(* Logix 5000 project; controller cal1615 1756-L62 rev 20.19; software revision 20.05; part 31 of 82 *)
(* tags used below, declared in another part *)
   FAULT : BOOL;   // Fault AFI
   p01_param_oven_timer_presets : DINT[32];   // System Parameter Oven Timer Presets
   p01_param_process_air_hl : REAL;   // Machine Parameter Process Air High Limit
   p01_sys_enc : SYS_ENC;   // System Encoder
   p01_sys_lc : Limit_Clamp;   // Zone 1 Misc Control Limit Clamp
   p01r09_pb_global_reset : BOOL;   // System Modes PB: Global Fault Reset
   p01r11 : routine;   // System Timer Presets
   p02_real_from_hmi : hmi_real;   // MOP HMI Iface Real from HMI
   p12r31_timer_warning : TIMER[5];   // Zone 2 Exhaust VFD Waringing Timer
   p12r32_timer_warning : TIMER[5];   // Zone 2 Supply VFD Warning Timer
   p13_di_exh_flow_ok : BOOL;   // Zone 3 Digital Input Exhaust Flow OK
   p13_di_recirc_flow_ok : BOOL;   // Zone 3 Digital Input Recirc Flow OK
   p13_param_fast_to_soak : REAL;   // Zone 3 Parameter Fast to Soak Control
   p13_param_lfl_hhl : REAL;   // Zone 3 Parameter High High Lower Flash Limit
   p13_param_lfl_hl : REAL;   // Zone 3 Parameter High LFL Limit
   p13_param_pid1_ff : REAL;   // Zone 3 Parameter Fast PID Bias
   p13_param_pid1_kd : REAL;   // Zone 3 Parameter Fast PID Derivative Gain
   p13_param_pid1_ki : REAL;   // Zone 3 Parameter Fast PID Integral Gain
   p13_param_pid1_kp : REAL;   // Zone 3 Parameter Fast PID Proportional Gain
   p13_param_pid2_ff : REAL;   // Zone 3 Parameter Auto PID Bias
   p13_param_pid2_kd : REAL;   // Zone 3 Parameter Auto PID Derivative Gain
   p13_param_pid2_ki : REAL;   // Zone 3 Parameter Auto PID Integral Gain
   p13_param_pid2_kp : REAL;   // Zone 3 Parameter Auto PID Proportional Gain
   p13_param_shutdown_temp : REAL;   // Zone 3 Parameter Zone Shutdown Temperature
   p13_param_soak_to_fast : REAL;   // Zone 3 Parameter Soak to Fast Control
   p13_param_tc01_dev : REAL;   // Zone 3 Parameter Oven Temperature Deviation from Setpoint
   p13_param_tc01_hl : REAL;   // Zone 3 Parameter Process Air High Limit
   p13_param_tc01z : REAL;   // Zone 3 Parameter Process Temperature Zero Offset
   p13_param_tc02z : REAL;   // Zone 3 Parameter SupplyTemperature Zero Offset
   p13_param_zone_pressure : REAL;   // Zone 3 Parameter High Pressure LImit
   p13r01 : routine;   // Zone 3 Main
   p13r02_timer_safe_temp : TIMER[2];   // Zone 3 Misc Control Chamber SafeTemperature Dwell
   p13r02_timer_warning : TIMER[4];   // Zone 3 Misc Control Warning Delay
   p13r09 : routine;   // Zone 3 Modes
   p13r09_timer_fault : TIMER[4];   // Zone 3 Modes Fault Delay
   p13r09_timer_warning : TIMER[8];   // Zone 3 Modes Warning Delay
   p13r10 : routine;   // Zone 3
   p13r10_timer_fault : TIMER[4];   // Zone 3 Fault Delay
   p13r10_timer_warning : TIMER[4];   // Zone 3 Warning Delay
   p13r20 : routine;   // Zone 3 Temp Sequence
   p13r20_state : DINT;   // Zone 3 Temperature Control State
   p13r20_status : DINT;   // Zone 3 Temperature Control Sequence Status
   p13r20_timer_fault : TIMER[4];   // Zone 3 Temp Sequence Fault Delay
   p13r20_timer_state_11 : TIMER;   // Zone 3 Temp Sequence State 11 Dwell
   p13r20_timer_state_3 : TIMER;   // Zone 3 Temperature Control State 3 Dwell
   p13r20_timer_state_4 : TIMER;   // Zone 3 Temp Sequence State 4 Dwell
   p13r20_timer_state_7 : TIMER;   // Zone 3 Temp Sequence State 7 Dwell
   p13r20_timer_warning : TIMER[4];   // Zone 3 Temp Sequence Warning Delay
   p13r30_cv_man_sp : REAL;   // Zone 3 Temperature Control Manual Heat Control Valve Setpoint
   p13r30_request_cool : BOOL;   // Zone 3 Temperature Control Request Cooling
   p13r30_request_manual : BOOL;   // Zone 3 Temperature Control Request Manual Control
   p13r30_temp_deviation_setpoint : DINT;
   p13r30_timer_fault : TIMER[16];   // Zone 3 Temperature Control Fault Delay
   p13r30_timer_warning : TIMER[12];   // Zone 3 Temperature Control Warning Delay
   p13r31_timer_fault : TIMER[5];   // Zone 3 Exhaust VFD Fault Timer
   p13r31_timer_warning : TIMER[5];   // Zone 3 Exhaust VFD Waringing Timer
   p13r32_timer_fault : TIMER[5];   // Zone 3 Recirc VFD Fault Timer
   p13r32_timer_warning : TIMER[5];   // Zone 3 Supply VFD Warning Timer
(* P13_Zone_3, continued *)

ROUTINE R09_Modes   (* ladder *)
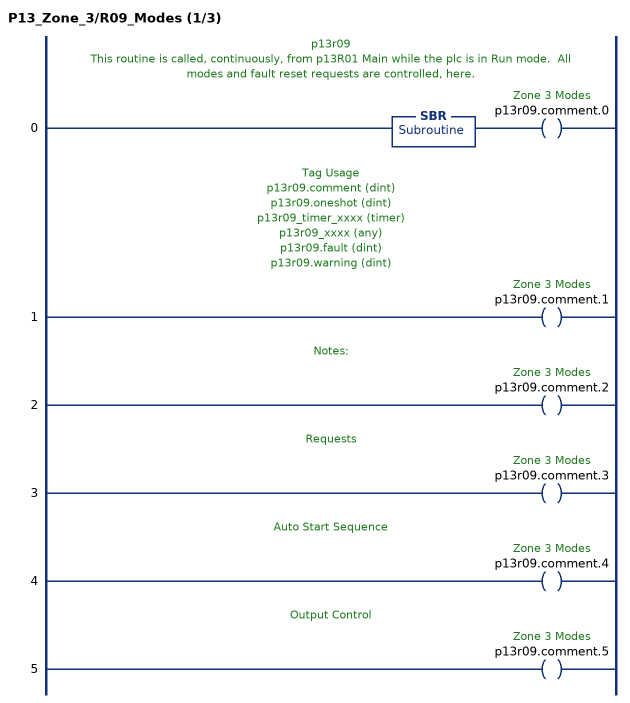
   // p13r09
   // This routine is called, continuously, from p13R01 Main while the plc is in Run mode.  All modes and fault reset requests are controlled, here.
   0: SBR()OTE(p13r09.comment.0);
   // Tag Usage
   // p13r09.comment (dint)
   // p13r09.oneshot (dint)
   // p13r09_timer_xxxx (timer)
   // p13r09_xxxx (any)
   // p13r09.fault (dint)
   // p13r09.warning (dint)
   1: OTE(p13r09.comment.1);
   // Notes:
   2: OTE(p13r09.comment.2);
   // Requests
   3: OTE(p13r09.comment.3);
   // Auto Start Sequence
   4: OTE(p13r09.comment.4);
   // Output Control
   5: OTE(p13r09.comment.5);
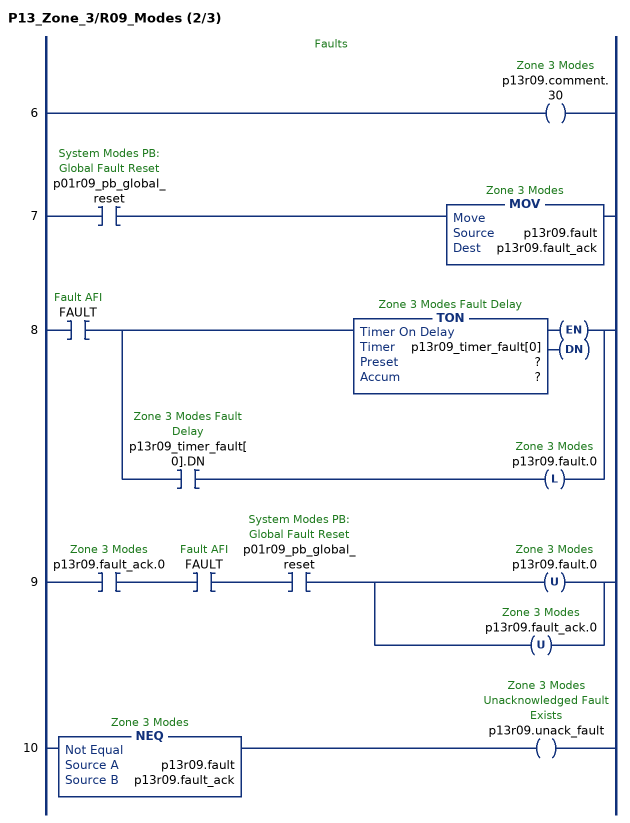
   // Faults
   6: OTE(p13r09.comment.30);
   7: XIC(p01r09_pb_global_reset)MOV(p13r09.fault,p13r09.fault_ack);
   8: XIC(FAULT)[TON(p13r09_timer_fault[0],?,?) ,XIC(p13r09_timer_fault[0].DN) OTL(p13r09.fault.0) ];
   9: XIC(p13r09.fault_ack.0)XIC(FAULT)XIC(p01r09_pb_global_reset)[OTU(p13r09.fault.0) ,OTU(p13r09.fault_ack.0) ];
   10: NEQ(p13r09.fault,p13r09.fault_ack)OTE(p13r09.unack_fault);
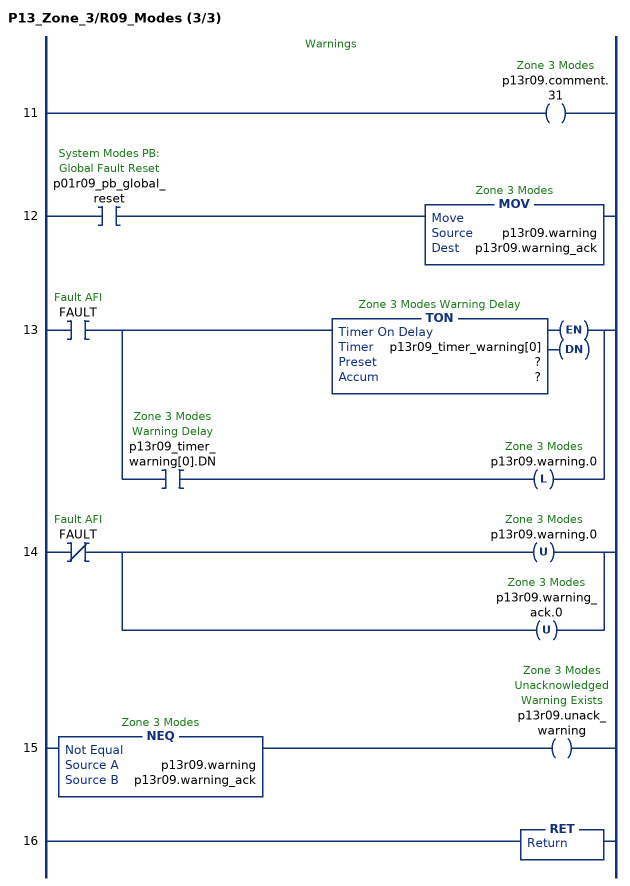
   // Warnings
   11: OTE(p13r09.comment.31);
   12: XIC(p01r09_pb_global_reset)MOV(p13r09.warning,p13r09.warning_ack);
   13: XIC(FAULT)[TON(p13r09_timer_warning[0],?,?) ,XIC(p13r09_timer_warning[0].DN) OTL(p13r09.warning.0) ];
   14: XIO(FAULT)[OTU(p13r09.warning.0) ,OTU(p13r09.warning_ack.0) ];
   15: NEQ(p13r09.warning,p13r09.warning_ack)OTE(p13r09.unack_warning);
   16: RET();
END_ROUTINE

ROUTINE R10_Parameters   (* ladder *)
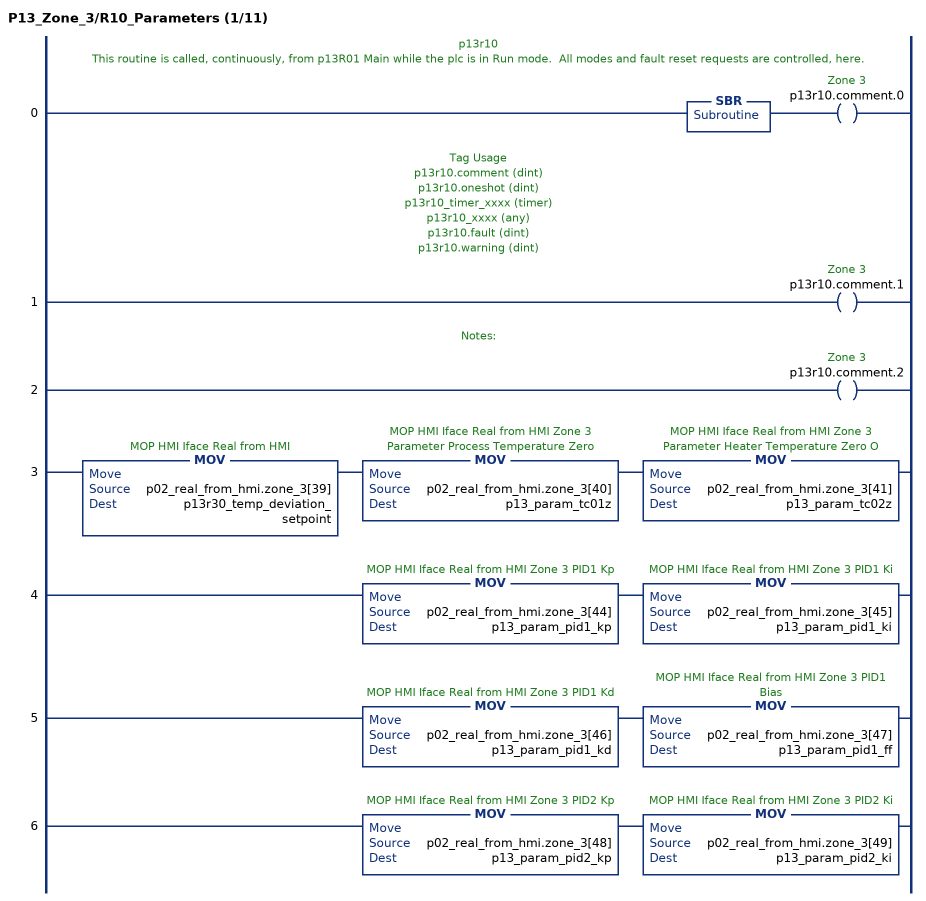
   // p13r10
   // This routine is called, continuously, from p13R01 Main while the plc is in Run mode.  All modes and fault reset requests are controlled, here.
   0: SBR()OTE(p13r10.comment.0);
   // Tag Usage
   // p13r10.comment (dint)
   // p13r10.oneshot (dint)
   // p13r10_timer_xxxx (timer)
   // p13r10_xxxx (any)
   // p13r10.fault (dint)
   // p13r10.warning (dint)
   1: OTE(p13r10.comment.1);
   // Notes:
   2: OTE(p13r10.comment.2);
   3: MOV(p02_real_from_hmi.zone_3[39],p13r30_temp_deviation_setpoint)MOV(p02_real_from_hmi.zone_3[40],p13_param_tc01z)MOV(p02_real_from_hmi.zone_3[41],p13_param_tc02z);
   4: MOV(p02_real_from_hmi.zone_3[44],p13_param_pid1_kp)MOV(p02_real_from_hmi.zone_3[45],p13_param_pid1_ki);
   5: MOV(p02_real_from_hmi.zone_3[46],p13_param_pid1_kd)MOV(p02_real_from_hmi.zone_3[47],p13_param_pid1_ff);
   6: MOV(p02_real_from_hmi.zone_3[48],p13_param_pid2_kp)MOV(p02_real_from_hmi.zone_3[49],p13_param_pid2_ki);
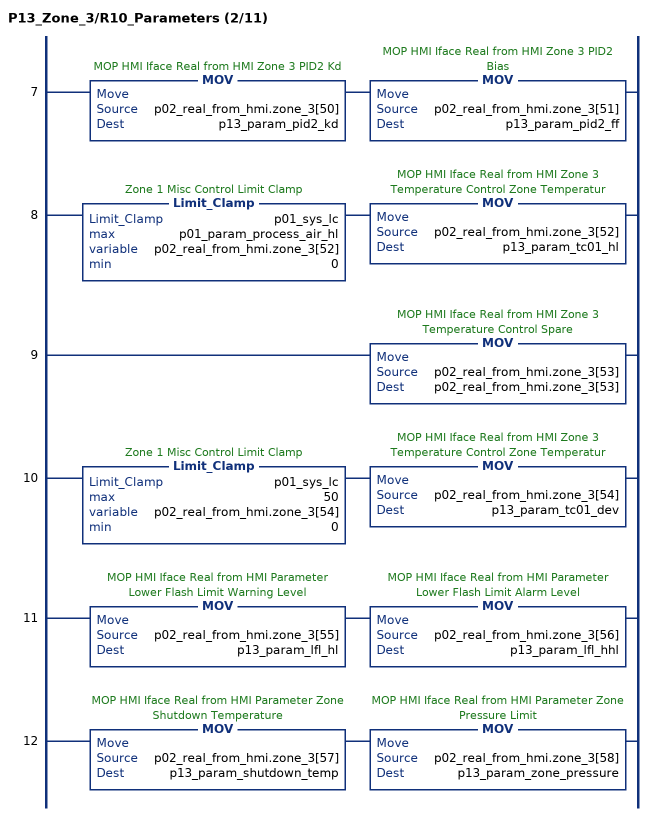
   7: MOV(p02_real_from_hmi.zone_3[50],p13_param_pid2_kd)MOV(p02_real_from_hmi.zone_3[51],p13_param_pid2_ff);
   8: Limit_Clamp(p01_sys_lc,p01_param_process_air_hl,p02_real_from_hmi.zone_3[52],0)MOV(p02_real_from_hmi.zone_3[52],p13_param_tc01_hl);
   9: MOV(p02_real_from_hmi.zone_3[53],p02_real_from_hmi.zone_3[53]);
   10: Limit_Clamp(p01_sys_lc,50,p02_real_from_hmi.zone_3[54],0)MOV(p02_real_from_hmi.zone_3[54],p13_param_tc01_dev);
   11: MOV(p02_real_from_hmi.zone_3[55],p13_param_lfl_hl)MOV(p02_real_from_hmi.zone_3[56],p13_param_lfl_hhl);
   12: MOV(p02_real_from_hmi.zone_3[57],p13_param_shutdown_temp)MOV(p02_real_from_hmi.zone_3[58],p13_param_zone_pressure);
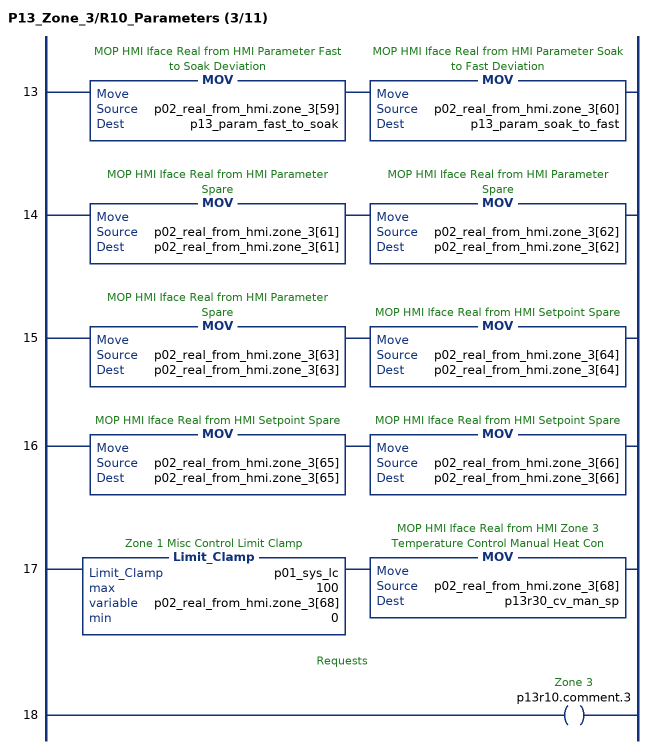
   13: MOV(p02_real_from_hmi.zone_3[59],p13_param_fast_to_soak)MOV(p02_real_from_hmi.zone_3[60],p13_param_soak_to_fast);
   14: MOV(p02_real_from_hmi.zone_3[61],p02_real_from_hmi.zone_3[61])MOV(p02_real_from_hmi.zone_3[62],p02_real_from_hmi.zone_3[62]);
   15: MOV(p02_real_from_hmi.zone_3[63],p02_real_from_hmi.zone_3[63])MOV(p02_real_from_hmi.zone_3[64],p02_real_from_hmi.zone_3[64]);
   16: MOV(p02_real_from_hmi.zone_3[65],p02_real_from_hmi.zone_3[65])MOV(p02_real_from_hmi.zone_3[66],p02_real_from_hmi.zone_3[66]);
   17: Limit_Clamp(p01_sys_lc,100,p02_real_from_hmi.zone_3[68],0)MOV(p02_real_from_hmi.zone_3[68],p13r30_cv_man_sp);
   // Requests
   18: OTE(p13r10.comment.3);
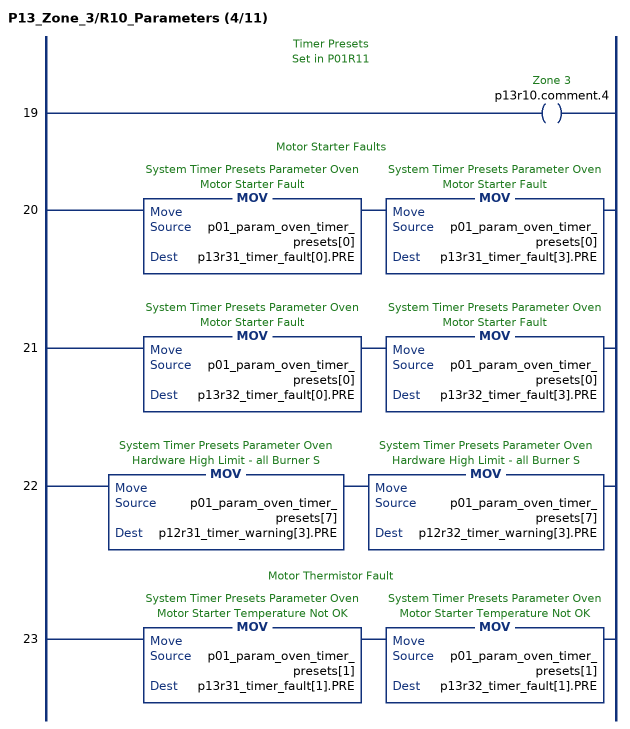
   // Timer Presets
   // Set in P01R11
   19: OTE(p13r10.comment.4);
   // Motor Starter Faults
   20: MOV(p01_param_oven_timer_presets[0],p13r31_timer_fault[0].PRE)MOV(p01_param_oven_timer_presets[0],p13r31_timer_fault[3].PRE);
   21: MOV(p01_param_oven_timer_presets[0],p13r32_timer_fault[0].PRE)MOV(p01_param_oven_timer_presets[0],p13r32_timer_fault[3].PRE);
   22: MOV(p01_param_oven_timer_presets[7],p12r31_timer_warning[3].PRE)MOV(p01_param_oven_timer_presets[7],p12r32_timer_warning[3].PRE);
   // Motor Thermistor Fault
   23: MOV(p01_param_oven_timer_presets[1],p13r31_timer_fault[1].PRE)MOV(p01_param_oven_timer_presets[1],p13r32_timer_fault[1].PRE);
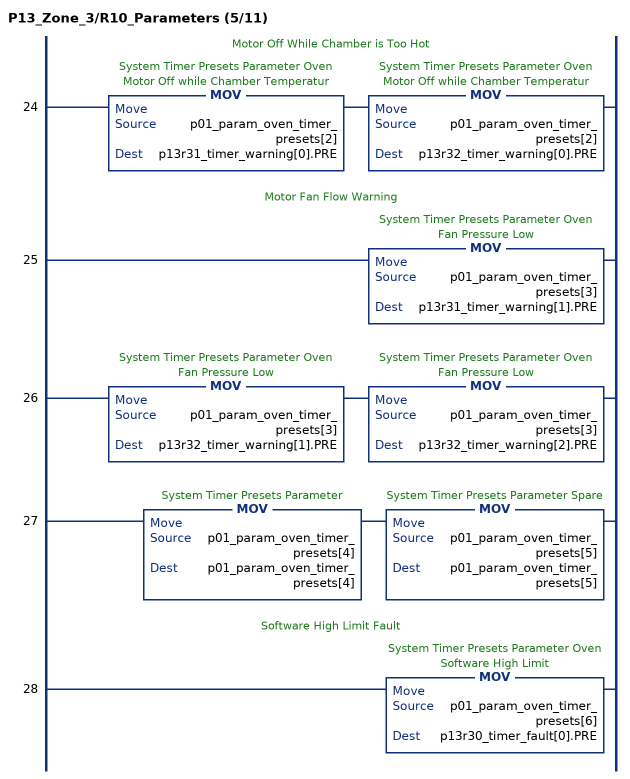
   // Motor Off While Chamber is Too Hot
   24: MOV(p01_param_oven_timer_presets[2],p13r31_timer_warning[0].PRE)MOV(p01_param_oven_timer_presets[2],p13r32_timer_warning[0].PRE);
   // Motor Fan Flow Warning
   25: MOV(p01_param_oven_timer_presets[3],p13r31_timer_warning[1].PRE);
   26: MOV(p01_param_oven_timer_presets[3],p13r32_timer_warning[1].PRE)MOV(p01_param_oven_timer_presets[3],p13r32_timer_warning[2].PRE);
   27: MOV(p01_param_oven_timer_presets[4],p01_param_oven_timer_presets[4])MOV(p01_param_oven_timer_presets[5],p01_param_oven_timer_presets[5]);
   // Software High Limit Fault
   28: MOV(p01_param_oven_timer_presets[6],p13r30_timer_fault[0].PRE);
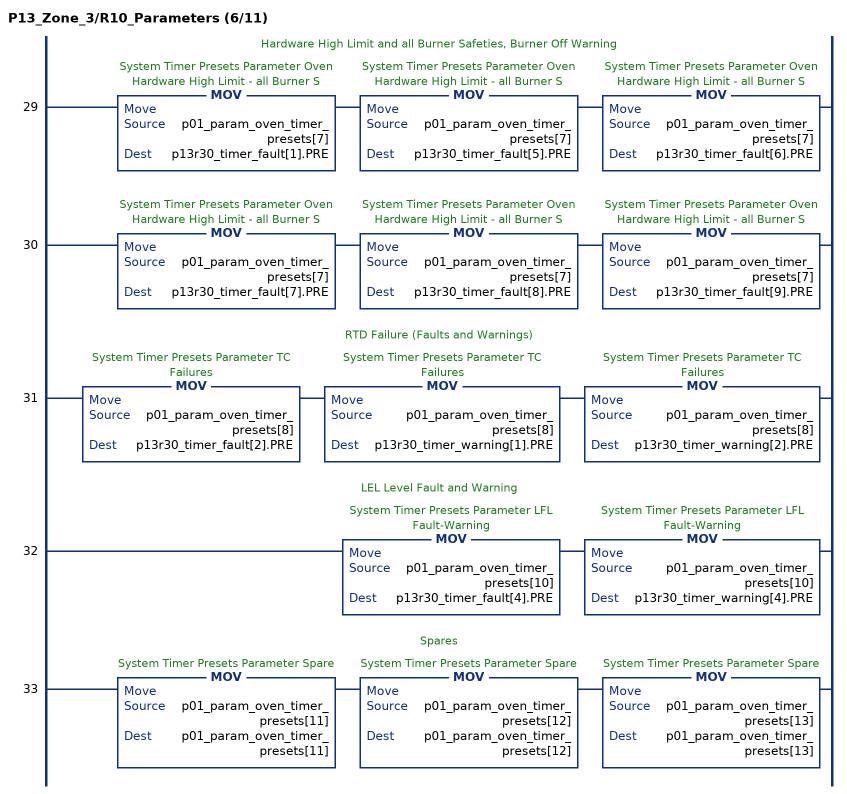
   // Hardware High Limit and all Burner Safeties, Burner Off Warning
   29: MOV(p01_param_oven_timer_presets[7],p13r30_timer_fault[1].PRE)MOV(p01_param_oven_timer_presets[7],p13r30_timer_fault[5].PRE)MOV(p01_param_oven_timer_presets[7],p13r30_timer_fault[6].PRE);
   30: MOV(p01_param_oven_timer_presets[7],p13r30_timer_fault[7].PRE)MOV(p01_param_oven_timer_presets[7],p13r30_timer_fault[8].PRE)MOV(p01_param_oven_timer_presets[7],p13r30_timer_fault[9].PRE);
   // RTD Failure (Faults and Warnings)
   31: MOV(p01_param_oven_timer_presets[8],p13r30_timer_fault[2].PRE)MOV(p01_param_oven_timer_presets[8],p13r30_timer_warning[1].PRE)MOV(p01_param_oven_timer_presets[8],p13r30_timer_warning[2].PRE);
   // LEL Level Fault and Warning
   32: MOV(p01_param_oven_timer_presets[10],p13r30_timer_fault[4].PRE)MOV(p01_param_oven_timer_presets[10],p13r30_timer_warning[4].PRE);
   // Spares
   33: MOV(p01_param_oven_timer_presets[11],p01_param_oven_timer_presets[11])MOV(p01_param_oven_timer_presets[12],p01_param_oven_timer_presets[12])MOV(p01_param_oven_timer_presets[13],p01_param_oven_timer_presets[13]);
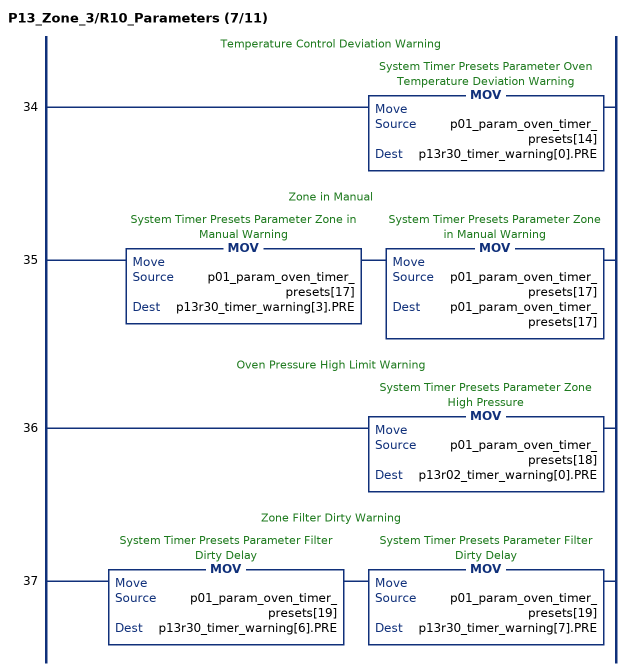
   // Temperature Control Deviation Warning
   34: MOV(p01_param_oven_timer_presets[14],p13r30_timer_warning[0].PRE);
   // Zone in Manual
   35: MOV(p01_param_oven_timer_presets[17],p13r30_timer_warning[3].PRE)MOV(p01_param_oven_timer_presets[17],p01_param_oven_timer_presets[17]);
   // Oven Pressure High Limit Warning
   36: MOV(p01_param_oven_timer_presets[18],p13r02_timer_warning[0].PRE);
   // Zone Filter Dirty Warning
   37: MOV(p01_param_oven_timer_presets[19],p13r30_timer_warning[6].PRE)MOV(p01_param_oven_timer_presets[19],p13r30_timer_warning[7].PRE);
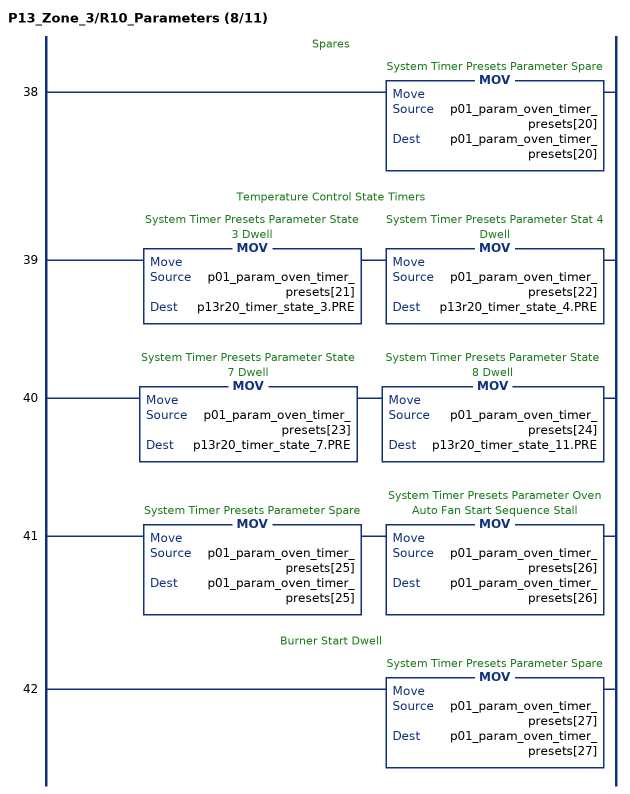
   // Spares
   38: MOV(p01_param_oven_timer_presets[20],p01_param_oven_timer_presets[20]);
   // Temperature Control State Timers
   39: MOV(p01_param_oven_timer_presets[21],p13r20_timer_state_3.PRE)MOV(p01_param_oven_timer_presets[22],p13r20_timer_state_4.PRE);
   40: MOV(p01_param_oven_timer_presets[23],p13r20_timer_state_7.PRE)MOV(p01_param_oven_timer_presets[24],p13r20_timer_state_11.PRE);
   41: MOV(p01_param_oven_timer_presets[25],p01_param_oven_timer_presets[25])MOV(p01_param_oven_timer_presets[26],p01_param_oven_timer_presets[26]);
   // Burner Start Dwell
   42: MOV(p01_param_oven_timer_presets[27],p01_param_oven_timer_presets[27]);
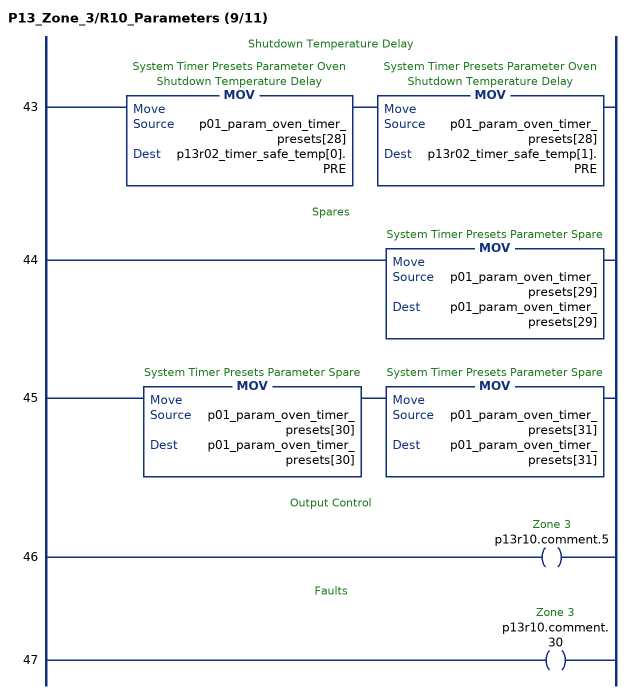
   // Shutdown Temperature Delay
   43: MOV(p01_param_oven_timer_presets[28],p13r02_timer_safe_temp[0].PRE)MOV(p01_param_oven_timer_presets[28],p13r02_timer_safe_temp[1].PRE);
   // Spares
   44: MOV(p01_param_oven_timer_presets[29],p01_param_oven_timer_presets[29]);
   45: MOV(p01_param_oven_timer_presets[30],p01_param_oven_timer_presets[30])MOV(p01_param_oven_timer_presets[31],p01_param_oven_timer_presets[31]);
   // Output Control
   46: OTE(p13r10.comment.5);
   // Faults
   47: OTE(p13r10.comment.30);
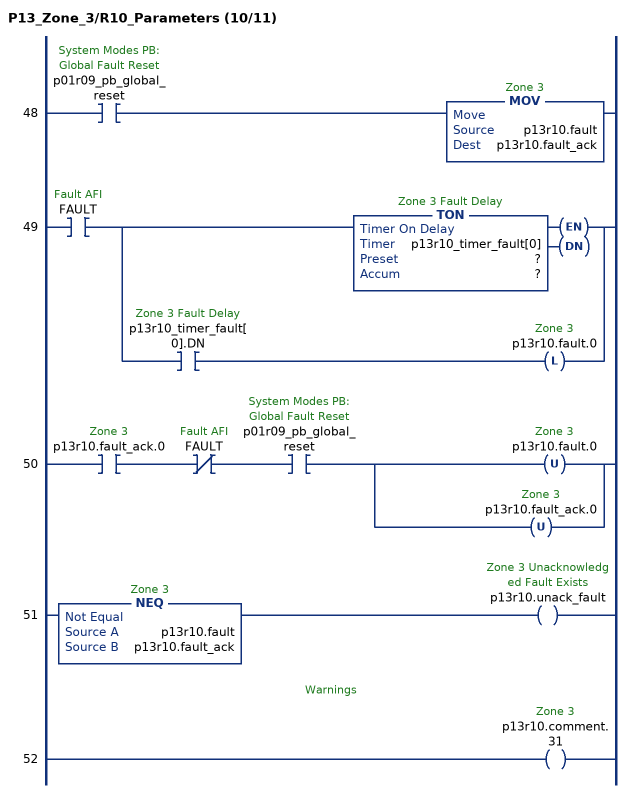
   48: XIC(p01r09_pb_global_reset)MOV(p13r10.fault,p13r10.fault_ack);
   49: XIC(FAULT)[TON(p13r10_timer_fault[0],?,?) ,XIC(p13r10_timer_fault[0].DN) OTL(p13r10.fault.0) ];
   50: XIC(p13r10.fault_ack.0)XIO(FAULT)XIC(p01r09_pb_global_reset)[OTU(p13r10.fault.0) ,OTU(p13r10.fault_ack.0) ];
   51: NEQ(p13r10.fault,p13r10.fault_ack)OTE(p13r10.unack_fault);
   // Warnings
   52: OTE(p13r10.comment.31);
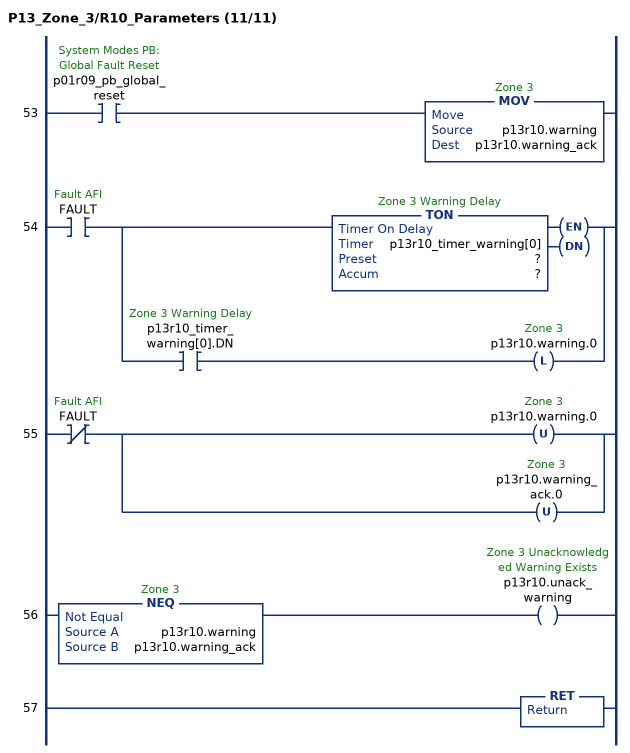
   53: XIC(p01r09_pb_global_reset)MOV(p13r10.warning,p13r10.warning_ack);
   54: XIC(FAULT)[TON(p13r10_timer_warning[0],?,?) ,XIC(p13r10_timer_warning[0].DN) OTL(p13r10.warning.0) ];
   55: XIO(FAULT)[OTU(p13r10.warning.0) ,OTU(p13r10.warning_ack.0) ];
   56: NEQ(p13r10.warning,p13r10.warning_ack)OTE(p13r10.unack_warning);
   57: RET();
END_ROUTINE

ROUTINE R20_Temp_Sequence   (* ladder *)
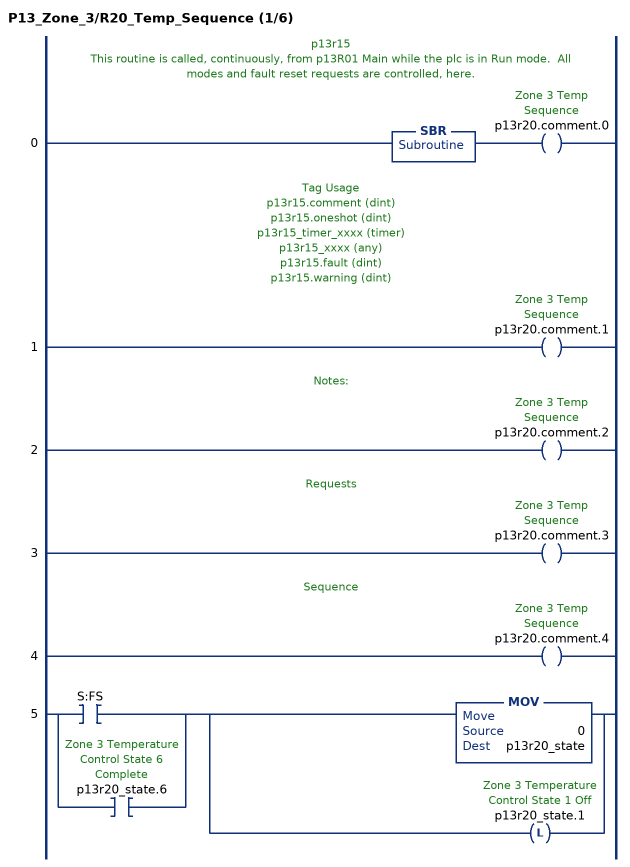
   // p13r15
   // This routine is called, continuously, from p13R01 Main while the plc is in Run mode.  All modes and fault reset requests are controlled, here.
   0: SBR()OTE(p13r20.comment.0);
   // Tag Usage
   // p13r15.comment (dint)
   // p13r15.oneshot (dint)
   // p13r15_timer_xxxx (timer)
   // p13r15_xxxx (any)
   // p13r15.fault (dint)
   // p13r15.warning (dint)
   1: OTE(p13r20.comment.1);
   // Notes:
   2: OTE(p13r20.comment.2);
   // Requests
   3: OTE(p13r20.comment.3);
   // Sequence
   4: OTE(p13r20.comment.4);
   5: [XIC(S:FS) ,XIC(p13r20_state.6) ][MOV(0,p13r20_state) ,OTL(p13r20_state.1) ];
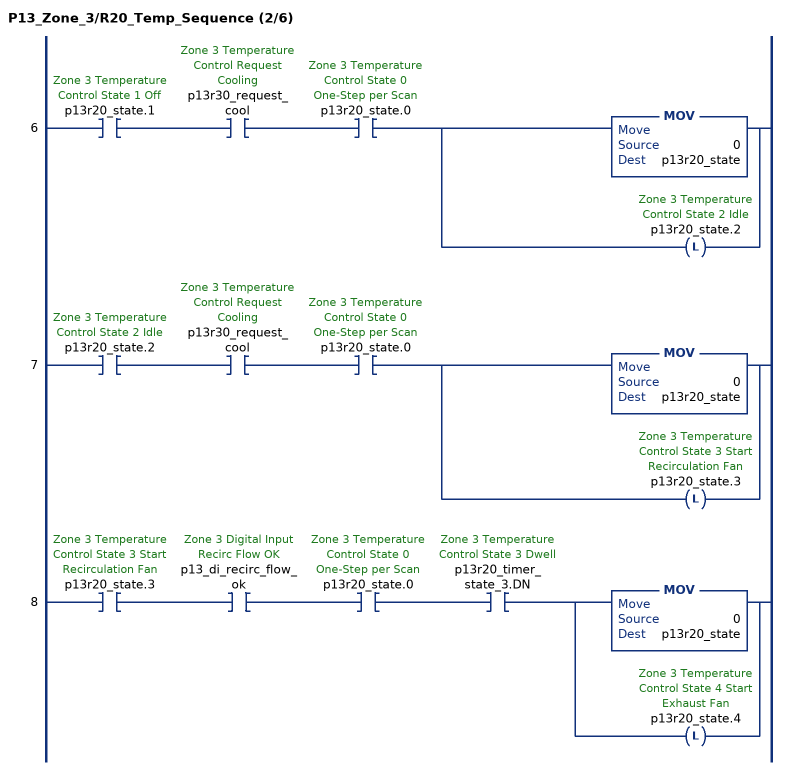
   6: XIC(p13r20_state.1)XIC(p13r30_request_cool)XIC(p13r20_state.0)[MOV(0,p13r20_state) ,OTL(p13r20_state.2) ];
   7: XIC(p13r20_state.2)XIC(p13r30_request_cool)XIC(p13r20_state.0)[MOV(0,p13r20_state) ,OTL(p13r20_state.3) ];
   8: XIC(p13r20_state.3)XIC(p13_di_recirc_flow_ok)XIC(p13r20_state.0)XIC(p13r20_timer_state_3.DN)[MOV(0,p13r20_state) ,OTL(p13r20_state.4) ];
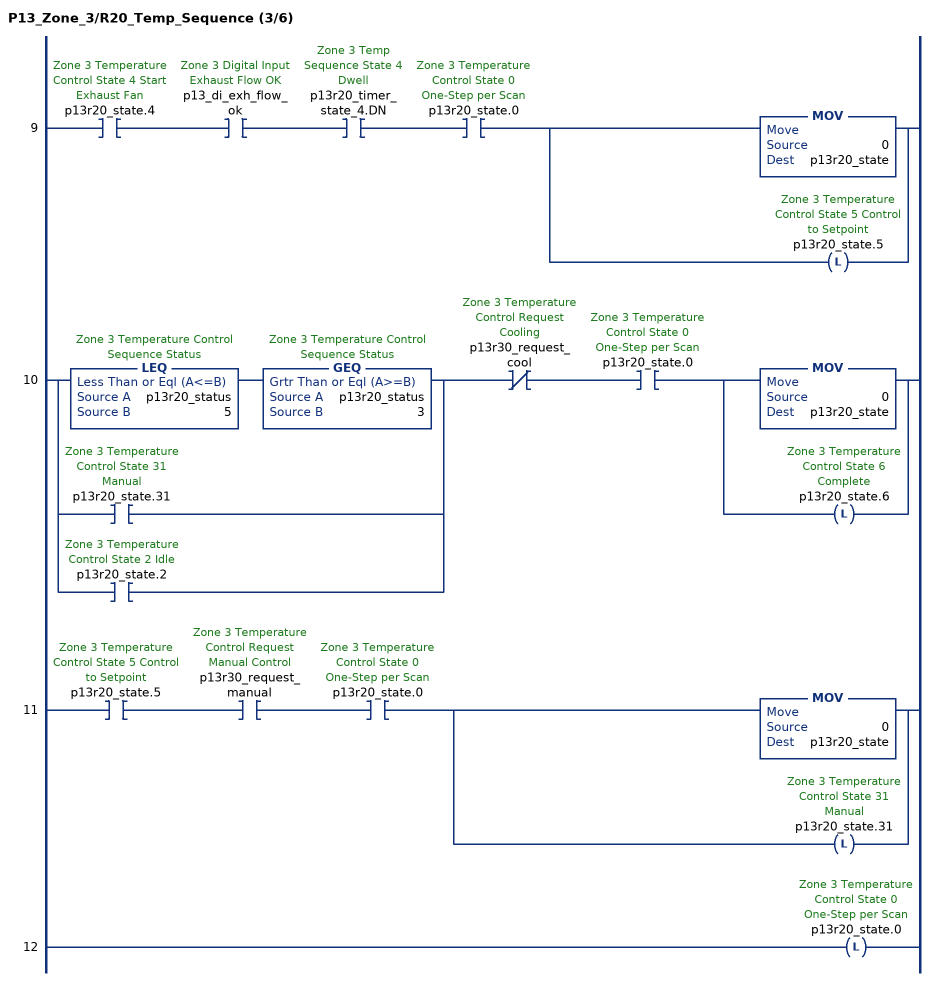
   9: XIC(p13r20_state.4)XIC(p13_di_exh_flow_ok)XIC(p13r20_timer_state_4.DN)XIC(p13r20_state.0)[MOV(0,p13r20_state) ,OTL(p13r20_state.5) ];
   10: [[LEQ(p13r20_status,5) GEQ(p13r20_status,3) ,XIC(p13r20_state.31) ] ,XIC(p13r20_state.2) ]XIO(p13r30_request_cool)XIC(p13r20_state.0)[MOV(0,p13r20_state) ,OTL(p13r20_state.6) ];
   11: XIC(p13r20_state.5)XIC(p13r30_request_manual)XIC(p13r20_state.0)[MOV(0,p13r20_state) ,OTL(p13r20_state.31) ];
   12: OTL(p13r20_state.0);
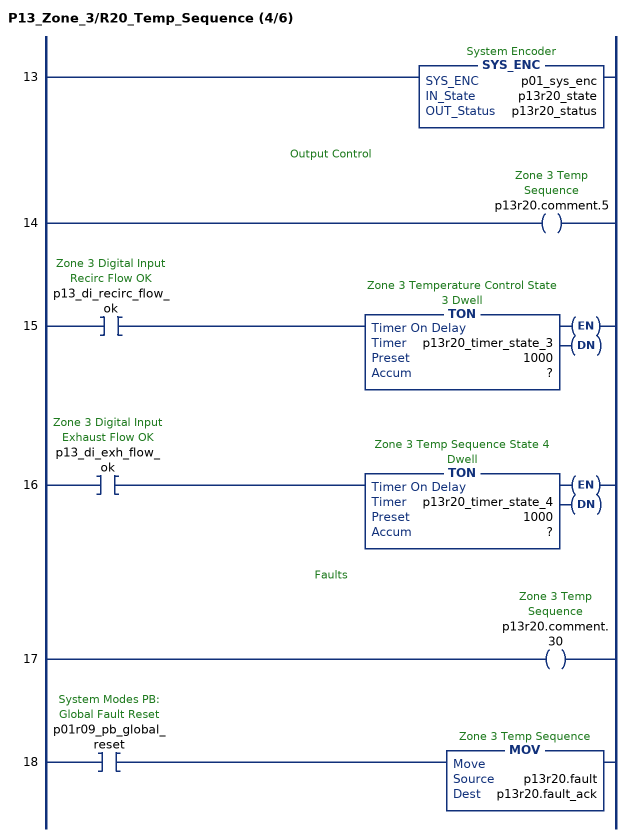
   13: SYS_ENC(p01_sys_enc,p13r20_state,p13r20_status);
   // Output Control
   14: OTE(p13r20.comment.5);
   15: XIC(p13_di_recirc_flow_ok)TON(p13r20_timer_state_3,?,?);
   16: XIC(p13_di_exh_flow_ok)TON(p13r20_timer_state_4,?,?);
   // Faults
   17: OTE(p13r20.comment.30);
   18: XIC(p01r09_pb_global_reset)MOV(p13r20.fault,p13r20.fault_ack);
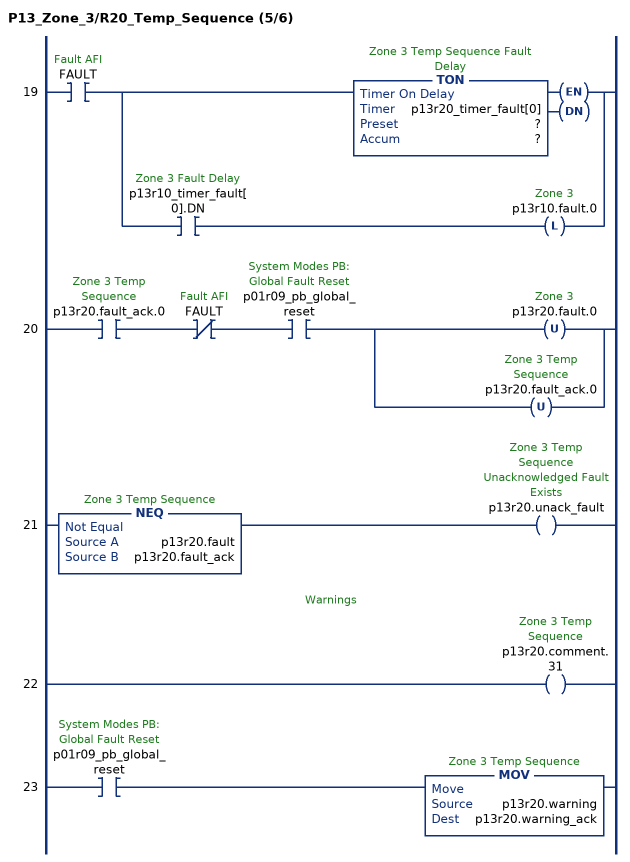
   19: XIC(FAULT)[TON(p13r20_timer_fault[0],?,?) ,XIC(p13r10_timer_fault[0].DN) OTL(p13r10.fault.0) ];
   20: XIC(p13r20.fault_ack.0)XIO(FAULT)XIC(p01r09_pb_global_reset)[OTU(p13r20.fault.0) ,OTU(p13r20.fault_ack.0) ];
   21: NEQ(p13r20.fault,p13r20.fault_ack)OTE(p13r20.unack_fault);
   // Warnings
   22: OTE(p13r20.comment.31);
   23: XIC(p01r09_pb_global_reset)MOV(p13r20.warning,p13r20.warning_ack);
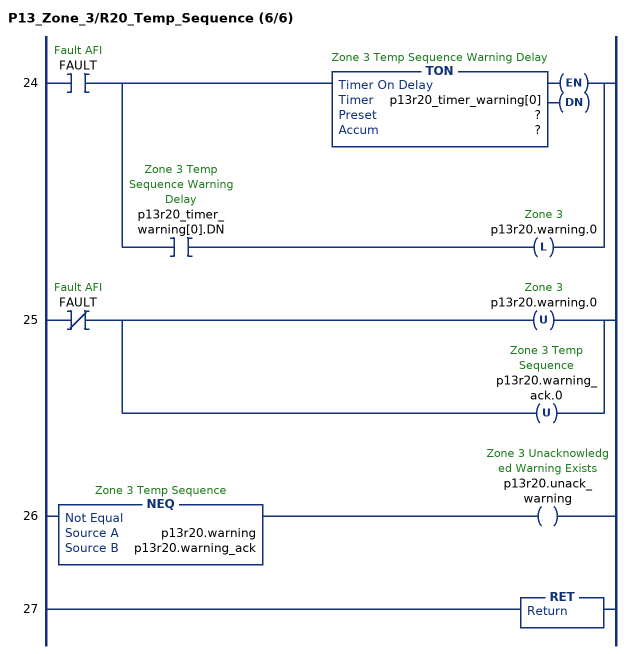
   24: XIC(FAULT)[TON(p13r20_timer_warning[0],?,?) ,XIC(p13r20_timer_warning[0].DN) OTL(p13r20.warning.0) ];
   25: XIO(FAULT)[OTU(p13r20.warning.0) ,OTU(p13r20.warning_ack.0) ];
   26: NEQ(p13r20.warning,p13r20.warning_ack)OTE(p13r20.unack_warning);
   27: RET();
END_ROUTINE
